FUNCTION F_LinkAlarm : BOOL
VAR_INPUT
//	bRaise				:BOOL;							//アラーム発生			インターフェースポインターが空だと困るのでコメントアウト
	bConfirm			:BOOL;							//アラーム確認
	bClear				:BOOL;							//アラームクリア
	bTrigger			:BOOL;							//アラーム発報条件
	ipResultMessage		:I_TcMessage;					//アラームメッセージ(I_TcMessage)
	fbAlarm				:REFERENCE TO FB_Alarm;			//アラーム(REFERENCE)
END_VAR
VAR
END_VAR

IF bTrigger=TRUE AND ipResultMessage<>0 AND fbAlarm.bRaised=FALSE THEN
	
	fbAlarm.CreateEx(stEventEntry := ipResultMessage.stEventEntry,TRUE, ipSourceInfo := ipResultMessage.ipSourceInfo);
	fbAlarm.bRaise:=TRUE;

ELSIF bTrigger=FALSE AND fbAlarm.bRaised=TRUE THEN

	fbAlarm.bConfirm:=bConfirm;
	
	fbAlarm.bClear:=bClear;

END_IF

fbAlarm();

END_FUNCTION

(* stored: Version 1.1.0.1, ProductVersion 3.1.4026.18
   POU F_LinkAlarm: Id {04abd3c1-b47e-4d4d-9b1c-983b50802c95}, SpecialFunc None *)
